Fanuc KAREL source: kd00072.KL

-- PROVISIONAL review KL for V1013-1; original PC SHA256 958f7ebf8cfd39ba219f6e1b323819fdac4f091395424a993e351ed816cd01e4
-- Incomplete behavior may be omitted. Consult companion uncertainty JSON. Do not deploy.
PROGRAM KD00072
%NOLOCKGROUP
VAR
  I : INTEGER
  J : INTEGER
  B : BOOLEAN
  R : REAL
  S : STRING[80]
BEGIN
  -- UNRESOLVED_PC offsets 5-13; opcodes 9D,2E,1F
  -- UNRESOLVED_PC offsets 18-22; opcodes 7F
END KD00072
